// TwinCAT 3 PLC project PLC
// ProgramVersion: 3.1.4023.0
// libraries:
//   Tc2_Standard, * (Beckhoff Automation GmbH)
//   Tc2_System, * (Beckhoff Automation GmbH)
//   Tc3_Module, * (Beckhoff Automation GmbH)
// project tree:
//   / PlcTask.TcTTO
//   POUs/ MAIN.TcPOU
// real-time tasks:
//   TASK PlcTask: cycle T#10ms, priority 20, ADS port 350

CONFIGURATION PLC
    RESOURCE PLC ON TwinCAT3
        TASK PlcTask(INTERVAL := T#10ms, PRIORITY := 20);
        PROGRAM MAIN WITH PlcTask : MAIN;
    END_RESOURCE
END_CONFIGURATION

// ---- POUs/MAIN.TcPOU
PROGRAM MAIN
VAR
	byteValue : BYTE := 255;
	wordValue : WORD :=	2300;
	dwordValue : DWORD := 10;
	sintValue : SINT := -50;
	intValue : INT := 16555;
	dintValue : DINT := 65345;
	realValue : REAL := 150.345;
	lrealValue : LREAL := - 50.50;
	myValue : BYTE := 1;
	myValue2 : DINT:=0;
END_VAR

END_PROGRAM
